Fanuc KAREL source: KT00693.KL

PROGRAM KT00693
%NOLOCKGROUP
VAR
  V1: VECTOR
  V2: VECTOR
  OUT: BOOLEAN
BEGIN
  V1.X = 1.0
  V2.Y = 2.0
  V1.X = 1.0
  V2.Y = 2.0
  OUT = + V1
END KT00693
